KUKA KRL program: C253_RESET_CICLO.src, C253_RESET_CICLO.dat

--- C253_RESET_CICLO.src ---
&ACCESS RV
&REL 3
DEF  C253_RESET_CICLO ( )
INTERRUPT OFF 1
BRAKE
WAIT FOR Program_PLC <> 99
INTERRUPT ON 1
END

--- C253_RESET_CICLO.dat ---
&ACCESS RV
&REL 3
DEFDAT C253_RESET_CICLO
;FOLD EXTERNAL DECLARATIONS;%{PE}%MKUKATPBASIS,%CEXT,%VCOMMON,%P
;FOLD BASISTECH EXT;%{PE}%MKUKATPBASIS,%CEXT,%VEXT,%P
EXT  BAS (BAS_COMMAND  :IN,REAL  :IN )
DECL INT SUCCESS
;ENDFOLD (BASISTECH EXT)
;FOLD USER EXT;%{E}%MKUKATPUSER,%CEXT,%VEXT,%P
;Make your modifications here

;ENDFOLD (USER EXT)
;ENDFOLD (EXTERNAL DECLARATIONS)
ENDDAT
